(*
Nazwa:			GVL
Opis:			Zmienne wykorzystywane globalnie
Wersja:			v0.2
Data:			2021-10-05
Autor:			DP,DJ
Urzadzenia:		
Konfiguracja:	
Info:
*)

//{attribute 'qualified_only'}

VAR_GLOBAL
	(******MAIN**********)
	//Ogólne
	bFirstCycle										:BOOL;									// Zmienna pierwszego cyklu
	bManualMode										:BOOL; (**)								// Włączony tryb serwisowy
	tMachineCycleTime								:TIME;									// Czas cyklu maszyny
	bAddGlobalCounter								:BOOL;									// Pomocnicza do dodawania licznika przy odrzucie	
	bAddBadPackageReason							:BOOL;
	bAddBadPackageReason2							:BOOL;
	bChangeover										:BOOL;		
	bPhaseChanging									:BOOL;									// Zmiana trybu na dwufazowy
	bBottleSorterDisable							:BOOL:=FALSE;
	bCapSorterDisable								:BOOL:=FALSE;	
	bFastSpeed										:BOOL;
	
	//Resetowanie 
	bCycleReseting									:BOOL;									//Resetowanie cyklu, trwa 1 sek
	bAllStationDoneDelay							:BOOL;
	bHomingDialog									:BOOL;									//Wyświetl komunikat o bazowaniu
	bHomingCanceled									:BOOL;									// Anulowano bazowanie
	bHoming											:BOOL;									// Trwa bazowanie
	bFirstPositioningDone							:BOOL;
	bRecipeChangePositioning						:BOOL;
	sHomingText										:STRING;
	bResetAfterErrorOrEstop							:BOOL;
	bResetStates									:BOOL;									//Reset cyklu i formatek
	//CycleLogic
	bRobotStationDone								:BOOL;									// Skonczyło się dozowanie lub wyłaczone
	nCheckWeiginhForm								:BOOL;
	//nExitWheelFormsTime							:UINT;									// Czas na wypuszczenie formatki z karuzeli jak pracuje transporter
	
	//Rejestry przesuwne
	bRFIDChecker									:BOOL;									// Sprawdzanie RFID
	bRFIDClearAfterRobot							:BOOL;									// Usuwanie numeru RFID za robotem
	iRFIDClearNr1AfterRobot							:INT;									// Usuwanie numeru RFID za robotem, usuniety = 0
	iRFIDClearNr2AfterRobot							:INT;									// Usuwanie numeru RFID za robotem, usuniety = 0
		
	eClearPackageState								:S_PackageState;
	
	eBottleFeederPackageState						:ARRAY [1..17] OF S_PackageState;		// [1..2] Struktura pod podajnikiem butelek

	eBeforeGatePackageState							:ARRAY [1..17] OF S_PackageState;		// [1..2] Struktura przed szlabane
	eBeforeDispencersPackageState					:ARRAY [1..17] OF S_PackageState;		// [1..4] Struktura przed dozownikami
	eDispencersPackageState							:ARRAY [1..17] OF S_PackageState;		// [1..4] Struktura pod dozownikami
	eAfterDispencersPackageState					:ARRAY [1..17] OF S_PackageState;		// [1..4] Struktura za dozownikami 
	eWeightPackageState								:ARRAY [1..17] OF S_PackageState;		// [1..5] Struktura nad wagami

	eBeforeLidFeeder2PackageState					:ARRAY [1..17] OF S_PackageState;		// [] Struktura przed podawaniem platynek
	eBeforeLidFeederPackageState					:ARRAY [1..17] OF S_PackageState;		// [] Struktura przed podawaniem platynek
	eLidFeederPackageState							:ARRAY [1..17] OF S_PackageState;		// [] Struktura podawania platynek
	eAfterLidFeederPackageState						:ARRAY [1..17] OF S_PackageState;		// [] Struktura przed podawaniem platynek
	eBeforeLidSealerPackageState					:ARRAY [1..17] OF S_PackageState;		// [] Struktura przed zgrzewaniem platynek
	eLidSealerPackageState							:ARRAY [1..17] OF S_PackageState;		// [] Struktura zgrzewanie platynek
	
	eBeforeGateCapSorterPackageState				:ARRAY [1..17] OF S_PackageState;		// [1..4] Struktura przed RFID sortera nasadek
	eBeforeCapSorterPackageState					:ARRAY [1..17] OF S_PackageState;		// [1..4] Struktura przed sorterem
	eCapSorterPackageState							:ARRAY [1..17] OF S_PackageState;		// [1..4] Struktura pod sorterem
	eAfterCapSorterPackageState						:ARRAY [1..17] OF S_PackageState;		// [1..4] Struktura za sorterem
	eBeforeCapControlPackageState					:ARRAY [1..17] OF S_PackageState;		// [1..1] Struktura pod sprawdzaniem obecnosci nakretki
	eBeforeScrewersPackageState						:ARRAY [1..17] OF S_PackageState;		// [1..6] Struktura przed zakręcarkami 
	eBeforeScrewers2PackageState					:ARRAY [1..17] OF S_PackageState;		// [1..6] Struktura przed zakręcarkami przed czujnikiem
	eUnderScrewerPackageState 						:ARRAY [1..17] OF S_PackageState;		// [1..3] Struktura pod zakręcarkami 
	eAfterScrewerPackageState						:ARRAY [1..17] OF S_PackageState;		// [1..8] Struktura za zakręcarkami 
	eUnderCorrectCapPackageState					:ARRAY [1..17] OF S_PackageState;		// [1..7] Struktura pomiedzy robotem a sprawdzeniem poprawnego zakrecenia
	eUnderCorrectCapPackageStateTemp				:ARRAY [1..17] OF S_PackageState;		// [1..7] Struktura pomiedzy robotem a sprawdzeniem poprawnego zakrecenia	
	eRobotPackageState								:ARRAY [1..17] OF S_PackageState;		// [1..2] Struktura pod robotem
	eHistoryPackageState							:ARRAY [1..1000] OF S_PackageState;		// Struktura historyczna przetransferowanych butelek
	eTempState1										:ARRAY [1..17] OF S_PackageState;		// [1..12] Za waga
	eTempState2										:ARRAY [1..17] OF S_PackageState;		// [1..12] Za podajnikiem butelek
	eTempState3										:ARRAY [1..17] OF S_PackageState;		// [1..12] Za sorterem nakretek	
	eRobotTempState									:ARRAY [1..17] OF S_PackageState;    	//  Pod robotem

	// Dodatkowe rejestry przy dozowaniu dwufazowyn
	
	eWeightPackage2PhasePackageState				:ARRAY [1..17] OF S_PackageState;		// [1..5] Struktura nad wagami (** dodane 07.04.2022**)
	eBeforeDispencer34PackageState2Phase			:ARRAY [1..17] OF S_PackageState;		// [1..5] Struktura nad wagami (** dodane 07.04.2022**)
	eDispencer34PackageState2Phase					:ARRAY [1..17] OF S_PackageState;		// [1..5] Struktura nad wagami (** dodane 07.04.2022**)
	eAfterDispencer34PackageState2Phase				:ARRAY [1..17] OF S_PackageState;		// [1..5] Struktura nad wagami (** dodane 07.04.2022**)
	eBeforeDispencer12PackageState2Phase			:ARRAY [1..17] OF S_PackageState;		// [1..5] Struktura nad wagami (** dodane 07.04.2022**)
	eDispencer12PackageState2Phase					:ARRAY [1..17] OF S_PackageState;		// [1..5] Struktura nad wagami (** dodane 07.04.2022**)
	eAfterDispencer12PackageState2Phase				:ARRAY [1..17] OF S_PackageState;		// [1..5] Struktura nad wagami (** dodane 07.04.2022**)

	(******P00_Alarms*****)

	AbActiveWarningDescription								:ARRAY [0..63] OF BOOL;	//  Aktywne ostrzeżenia	
	
	//Sygnał dzwiekowy
	bSoftAlarm										:BOOL;
	
	bResetError										:BOOL:=FALSE;(**)						// Zmienna resetująca stację/błąd w PLC ,wystawia się po wciśnięciu ResetVisuCmd			
	//Reset Diagnostyki	
	
	//Alarmy inne*
	GeneralAlarms									:S_Error;								// 1 Ogólne
	//*Alarmy Stacji
	FormTransporterDispencerError					:S_Error;								// 2 Transporter wwjazdowy pod dozowniki
	FormTransporterScrewerError						:S_Error;								// 2 Transporter wyjściowy
	FormTransporterROPPError						:S_Error;
	FormTransporterAfterCapSorterError				:S_Error;
	FormTransporterBeforeScrewerError				:S_Error; 								// 3 Transporrter przed zakręcarkami
	FormTransporterSlowerError						:S_Error; 								// Spowalniacz
	FormTransporterAfterScrewerError				:S_Error; 								// 3 Transporrter przed zakręcarkami
	FormTransporterAfterBottleTransferError			:S_Error; 								
	BottleFeederError								:S_Error;								// Podajnik butelek
	BottleFeederTurnTableError						:S_Error;								// Stół obrotowy podajnika butleek
	BottleFeederFormGateError						:S_Error;								// Stoper formatek
	PucksInserterError								:S_Error;								// Podajnik butelek
	PucksInserterTurnTableError						:S_Error;								// Stół obrotowy podajnika opakowań
	PucksInserterFormGateError						:S_Error;								// Stoper formatek
	PucksInserterPushTableError_m1					:S_Error;								//71U3
	PucksInserterPushTableError_m2					:S_Error;								//71U4
	PucksInserterPushTableError_m3					:S_Error;								//
	GateBeforeDispencersError						:S_Error;		   						// 3A Szlaban przed dozownikami
		

	BarrierBetweenDispencers						:S_Error;								// Obsługa błędów szlaban dozowniki ( dozowanie dwufazowe, pod dozownikamia);
	BarrierBetweenWeights							:S_Error;								// Obsługa błędów stacji szlabanu pomiedzy wagamia ( dozowanie dwufazowe, wjazd na wagi);
	
	// Alarm wyciągu
	
	ExhaustFanError									:S_Error;
	SensorAcetoneError								:S_Error;								// Obśługa błedów czujnika acetonu
	SensorAirFlowError								:S_Error;								// Obsługa błędów czujnika przepływu 
	
	BottlePusherError								:S_Error;	
	//DispencerGatesError							:S_Error;								// 4 Szlabany pod dozownikami
	DispencersDragLeftError							:S_Error;								// Przeciąganie formatek
	DispencersDragRightError						:S_Error;								// Przeciąganie formatek (** 15.04.22 Damian**)
	

	DispencersCatch1Error							:S_Error;								// 4 Chwytak butelek dozownika 1
	DispencersCatch2Error							:S_Error;								// 4 Chwytak butelek dozownika 2
	DispencersCatch3Error							:S_Error;								// 4 Chwytak butelek dozownika 3
	DispencersCatch4Error							:S_Error;								// 4 Chwytak butelek dozownika 4
	Dispencer1Error									:S_Error;								// 5 Dozownik nr 1
	Dispencer2Error									:S_Error;								// 6 Dozownik nr 2
	Dispencer3Error									:S_Error;								// 6 Dozownik nr 3	
	Dispencer4Error									:S_Error;								// 6 Dozownik nr 4		
	TankHeatingError								:S_Error;								// Grzanie zbiornka

	WeightLiftError									:S_Error;
	
	Weight1Error									:S_Error;								// 8 Waga pierwsza jednofazowe
	Weight2Error									:S_Error;								// 8 Waga druga jednofazowe
	Weight3Error									:S_Error;								// 8 Waga trzecia jednofazowe
	Weight4Error									:S_Error;								// 8 Waga czwarta jednofazowe
	Weight5Error									:S_Error;								// 8 Waga piąta jednofazowe   	(** dodane 07.04.2022**)
	Weight6Error									:S_Error;								// 8 Waga szósta jednofazowe	(** dodane 07.04.2022**)
	
	
	GateAfterWeightError							:S_Error;								// 9 Szlaban za wagamia
		
	Dispencer1CorrectionError						:S_Error;	
	Dispencer2CorrectionError						:S_Error;
	Dispencer3CorrectionError						:S_Error;	
	Dispencer4CorrectionError						:S_Error;	
	WickFeederSorterError							:S_Error;
	
	
	CapFeederError									:S_Error;								// 14 
	CapSorterDragError								:S_Error;								// 15  Przeciąganie pod sorterem nasadek
			
	CapPuttedCheckError								:S_Error;								// 17 Wykrycie zakrętki
	
	GripperScrewerCatch1Error						:S_Error;								// 18 Chwytak zakręcarki szczękowej
	GripperScrewerCatch2Error						:S_Error;								// 18 Chwytak zakręcarki szczękowej
	GripperScrewer1Error							:S_Error;								// 19 Zakręcerka szczękowa 1
	GripperScrewer2Error							:S_Error;								// 19 Zakręcerka szczękowa 1

	BottleDragError									:S_Error;								//19.1 Przeciąganie butelek pod zakręcarkami
	CapCorrectCheckError							:S_Error;								// 21B Sprawdzanie zakręconej nakrętki
	CapCorrectCheckCameraError						:S_Error;
	BottleTransferError								:S_Error;								// 22 Robot
	GateRobotError									:S_Error;								// 22 Szlabany pod robotem
	BottleTransferAfterDragError					:S_Error;								// 14 

	BadBottleConveyorError							:S_Error;								// 23 Transporter odrzuconych butelek	
	LabelMachineError								:S_Error;								// 24 Etykieciarka
	TanksError										:S_Error;								// 24 Zbiorniki
	ExitTurnTableError								:S_Error;								// 25 Stół odbierający
	ExitConveyorError								:S_Error;								// 


	BarrierLidFeeder								: S_Error;								// Podajnik platynek 
	LidFeederError									: S_Error;								// Podajnik platynek 
	LidFeeder2Error									: S_Error;								// Podajnik platynek 2
	LidFeederFormPositioningError					: S_Error;	
						
	BarrierWickFeeder								: S_Error;
	WickFeederDragError								: S_Error;
	WickFeederError									: S_Error;
	WickFeeder2Error								: S_Error;
	WickFeederFormPositioningError					: S_Error;
	
	LidFeederDragError								: S_Error;								// Przeciąganie formatek                                                                                          
	LidPuttedCheckError								: S_Error;								// Wykrycie platynki                                                                                         
	LidSealerError									: S_Error;								// Zgrzewarka 1
	LidSealer2Error									: S_Error;								// Zgrzewarka 2
	LidSealerDragError								: S_Error;								// Przeciąganie formatek
	
	
	
	
	//Warningi
	TanksWarning									:ARRAY [0..7] OF S_Warning;							
	BottleTransferWarning							:ARRAY [0..7] OF S_Warning;	
	GeneralWarning1									:ARRAY [0..7] OF S_Warning;
	WeightWarning									:ARRAY [0..7] OF S_Warning;		
	DispencersWarning								:ARRAY [0..7] OF S_Warning;		
	ScrewersWarning									:ARRAY [0..7] OF S_Warning;		
	BottleFeederWarning								:ARRAY [0..7] OF S_Warning;
	ExSensorWarning									:ARRAY [0..7] OF S_Warning;
	CapFeederWarning								:ARRAY [0..7] OF S_Warning;	
	CapSorterWarning								:ARRAY [0..7] OF S_Warning;		
	BottleSorterWarning								:ARRAY [0..7] OF S_Warning;	
	LidFeederWarning								:ARRAY [0..7] OF S_Warning;		
	WickFeederWarning								:ARRAY [0..7] OF S_Warning;	
	WickFeederSorterWarning							:ARRAY [0..7] OF S_Warning;	
	(********P00_OEE********)		
	udiCounterExecuteTimeTemp						:UDINT;
	udiCounterErrorTimeTemp							:UDINT;
	udiCounterReadyTimeTemp							:UDINT;

	
	(******P00_Basic*******)
	//impulsy
	bImp1Sec										:BOOL;									// Impuls na zbocze generatora 1 sek
	b1Hz											:BOOL;									// Generator 1 sekundowy
	bV1Hz											:BOOL;									// bit o czest. 1Hz
	b2Hz											:BOOL;									// Generator 0,5 sekundowy
	//czas
	dtActTime										:DT;
	wYear 											:WORD;
	wMonth											:WORD;
	wDayOfWeek 										:WORD;
	wDay 											:WORD;
	wHour 											:WORD;
	wMinute 										:WORD;
	wSecond 										:WORD;
	wMilliseconds 									:WORD;

	//Zmienne podst.
	bAlwaysFalse									:BOOL:=FALSE;							//Zawsze zero
	
	(*****P00_PneumaticsValves***)
	(*****Receptury****)	
	bVTEMEnable										:BOOL;
	lrGripperScrewerPressure						:LREAL;									//Ciśnienie siłownika chwytaka nasadki zakręcarki szczękowej 1 (0.0 kg)
	lrGripperScrewerPressureExhaustLevel			:LREAL;									//Prędkość zamykania siłownika chwytaka nasadki zakręcarki szczękowej 1 (0.0-100.0 %)
	lrGripperScrewerCatchPressure					:LREAL;									//Ciśnienie siłownika chwytaka butelki zakręcarki szczękowej 1 (0.0 kg)
	lrGripperScrewerCatchPressureExhaustLevel		:LREAL;									//Prędkość zamykania siłownika chwytaka butelki zakręcarki szczękowej 1 (0.0-100.0 %)
	lrDispencerCatchPressure						:LREAL;

	(*****P0_Recipes***)
	(*****Receptury****)
	sRecipeName										:STRING;				
	sRecipeIndex									:STRING;				
	nRecipeIndex									:REAL;					
	bRecipeAfterPowerStateChosen					:BOOL;									//Receptura w stanie Power została wybrana (Pierwsza receptura po uruchomieniu)
	iPackageCapType									:INT; 									// Typ nasadki 
	iPackageCapDiameter								:INT;
	
	//[H] Praca w trybie wybuchowym
	bExEnable										:BOOL;						// [H] Tryb EX
	
	
	(****P01_BottleFeeder****)
	bBottleFeederEnable								:BOOL;									// Zezwolenie na pracę stacji podawania opakowań
	bBottleFeederDoHoming							:BOOL;									// Wykonanie bazowania stacji podawania butelek
	bBottleFeederTurnTableRun						:BOOL;									// Komenda startu stołu obrotwego
	iBottleFeederBottleSensorDelay					:INT;
	iBottleFeederFormGateDelay						:INT;
	iBottleFeederAllowFormDelay						:INT;
	bBottleFeederFormGateRun						:BOOL;									// Bit sterujacy działanie bramki 
	iBottleFeederTurntableVelocitySV				:UDINT;	

	(****P01_PucksInserter****)
	bPucksInserterEnable							:BOOL;									// Zezwolenie na pracę stacji 
	bPucksInserterDoHoming							:BOOL;									// Wykonanie bazowania stacji 
	bPucksInserterTurnTableRun						:BOOL;									// Komenda startu stołu obrotwego
	iPucksInserterBottleSensorDelay					:INT;
	iPucksInserterFormGateDelay						:INT;
	iPucksInserterFormGateDelayAdd					:INT;	
	iPucksInserterAllowFormDelay					:INT;
	bPucksInserterFormGateRun						:BOOL;									// Bit sterujacy działanie bramki 
	iPucksInserterTurntableVelocitySV				:UDINT;	
	iPucksInserterConveyorVelocitySV				:UDINT;	
	aPucksInserterWheelAxisRef						:AXIS_REF;								// Struktura osi 
	lrPucksInserterWheelOffset						:LREAL;									// Offset karuzeli +-10 st.
	lrPucksInserterWheelAcceleration				:LREAL;									// Przyspieszenie 
	lrPucksInserterWheelVelocity					:LREAL;									// Prędkość 
	lrPucksInserterHammerHeightSV					:LREAL;									// Pozycja
	
	//Push table 27.05 Vasyl	
	bPucksInserterPushTable_m1_Enable					:BOOL;
	bPucksInserterPushTable_m1_Run						:BOOL;
	udiPucksInserterPushTable_m1_VelocitySV				:UDINT;
	bPucksInserterPushTable_m2_Enable					:BOOL;
	bPucksInserterPushTable_m2_Run						:BOOL;
	udiPucksInserterPushTable_m2_VelocitySV				:UDINT;
	bPucksInserterPushTable_m3_Enable					:BOOL;
	bPucksInserterPushTable_m3_Run						:BOOL;
	udiPucksInserterPushTable_m3_VelocitySV				:UDINT;

	udiPucksInserterPushTableActuatorPUSHDelay			:UDINT;
	udiPucksInserterPushTableActuatorPULLDelay			:UDINT;
	udiPucksInserterPushTableOFFDelay					:UDINT;

	(****P01_BottleSorter****)
	//Po komunikacji
	
	(*****P01_Gates********)
	bGateBeforeDispencersEnable						:BOOL;									//Zezwolenie na pracę szlabanów pod robotem
	nGateBeforeDispencersTimeFormInserting			:UINT;									//Czas od momentu wjazdu formatek do zamkniecia 1 szlabanu pod robotem
	
	bGateAfterWeightEnable							:BOOL;									//Zezwolenie na pracę szlabanów pod robotem
	nGateAfterWeightTimeFormInserting				:UINT;									//Czas od momentu wjazdu formatek do zamkniecia 1 szlabanu pod robotem
		
	bBarrierLidFeederEnable							:BOOL;									//Zezwolenie na pracę szlabanów pod robotem
	nBarrierLidFeederTimeFormInserting				:UINT;									//Czas od momentu wjazdu formatek do zamkniecia 1 szlabanu pod robotem
	
	bGateRobotEnable								:BOOL;									//Zezwolenie na pracę szlabanów pod robotem
	nGateRobotTimeFormInserting						:UINT;									//Czas od momentu wjazdu formatek do zamkniecia 1 szlabanu pod robotem
	
	(*****P01_Barriers********)
	bBarrierWeightRun								:BOOL;									// Komenda otwarcia bariery przed wagami
	bBarrierDispencerRun							:BOOL;									// Komenda otwarcia bariery przed wagami
	
	(*****P02_Dispencers***)
	bCIP											: BOOL; // Włączone mycie CIP
	bDispencer1Cleaning								: BOOL;	// Mycie dozowników
	bDispencer2Cleaning								: BOOL;	// Mycie dozowników
	bDispencer3Cleaning								: BOOL;	// Mycie dozowników
	bDispencer4Cleaning								: BOOL;	// Mycie dozowników

	bDispencer1DoSync								: BOOL;	// Ustawienie tłoka/podnośnika 1 dozownika na konkretną pozycję (otwierają się zawory ssania) tylko w trybie serwisowym 
	bDispencer2DoSync								: BOOL;	// Ustawienie tłoka/podnośnika 2 dozownika na konkretną pozycję (otwierają się zawory ssania) tylko w trybie serwisowym 
	bDispencer3DoSync								: BOOL;	// Ustawienie tłoka/podnośnika 3 dozownika na konkretną pozycję (otwierają się zawory ssania) tylko w trybie serwisowym 
	bDispencer4DoSync								: BOOL;	// Ustawienie tłoka/podnośnika 4 dozownika na konkretną pozycję (otwierają się zawory ssania) tylko w trybie serwisowym 

	//Dozowniki 
	bDispencer12AllowDosingAfterDrag				:BOOL;
	bDispencer34AllowDosingAfterDrag				:BOOL;	
	bDoorDispencerOpen								:BOOL;
	bDosingTwoPhases								:BOOL;									//Dozowanie dwu fazowe
	bDispencersDoHoming								:BOOL;									//Wykonanie bazowania dozowniki
    lrDispencersLifterReadyPosition					:LREAL;									//Pozycja podnonika przy której dozowniki są w stanie gotowości
	uiDispencerStartDosingDelay						:UINT;(*0-3000*)				 		// Czas opóźnienia rozpoczęcia dozowania

//	Dozownik 1
	aDispencer1AxisRef								:AXIS_REF;//ActPos	(**)				// Struktura osi dozownika 1
	aDispencerLifter12AxisRef						:AXIS_REF;//ActPos	(**)				// Struktura osi dozownika 1
	bDispencer1Enable								:BOOL; 									// Zezwolenie na prace dozownika 1
	lrDispencer1DoseVolume							:LREAL:=195; 							// Objętoć do wydozowania przez dozownik 1
	bDispencer1LiftSynchroPh1						:BOOL;						 			// Polecenie synchronizacji dozownika z podnonikiem w fazie 1 Dozownika 1
	bDispencer1LiftSynchroPh2						:BOOL; 					 				// Polecenie synchronizacji dozownika z podnonikiem w fazie 2 Dozownika 1
	bDispencer1LiftSynchroPh3						:BOOL; 									// Polecenie synchronizacji dozownika z podnonikiem w fazie 3 Dozownika 1
	lrDispencer1Phase1Volume						:LREAL:=100;							// Objętoć do której ma trwać faza pierwsza dozowania dozownika 1
	lrDispencer1Phase2Volume						:LREAL:=100;							// Objętoć do której ma trwać faza druga dozowania dozownika 1
	lrDispencer1Phase1Velocity						:LREAL:=500;							// Prędkoć z jakš ma byc wykonywana faza pierwsza dozowania dozownika 1
	lrDispencer1Phase2Velocity						:LREAL:=500;							// Prędkoć z jakš ma byc wykonywana faza druga dozowania dozownika 1
	lrDispencer1Phase3Velocity						:LREAL:=500;							// Prędkoć z jakš ma byc wykonywana faza trzecia dozowania dozownika 1
	lrDispencer1SuckVelocity						:LREAL:=500;							// Prędkoć z jakš ma byc wykonywane zasysanie dozownika 1
	lrDispencer1Phase1Acceleration					:LREAL:=3000;							// Przyspieszenie z jakim ma byc wykonywana faza 1  dozownika 1
	lrDispencer1Phase2Acceleration					:LREAL:=3000;							// Przyspieszenie z jakim ma byc wykonywana faza 2  dozownika 1
	lrDispencer1Phase3Acceleration					:LREAL:=3000;							// Przyspieszenie z jakim ma byc wykonywana faza 3  dozownika 1
	lrDispencer1SuckAcceleration					:LREAL:=3000;							// Przyspieszenie z jakim ma byc wykonywane zasysanie dozownika 1
	lrDispencer1Phase1Deceleration					:LREAL:=3000;							// Zwalnianie z jakim ma byc wykonywana faza 1  dozownika 1
	lrDispencer1Phase2Deceleration					:LREAL:=3000;							// Zwalnianie z jakim ma byc wykonywana faza 2  dozownika 1
	lrDispencer1Phase3Deceleration					:LREAL:=3000;							// Zwalnianie z jakim ma byc wykonywana faza 3  dozownika 1
	udiDispencer1DosingDoneDelayTime				:UDINT:=20; 							// Opóźnienie wykonania cyklu dozy przez dozownik 1 [ms]
	lrDispencer1SuckValveOpenVolume					:LREAL:=0;(*Z 0-15*)					//[3] Objętość przy której ma byc otwierany zawór ssania dozownika 1
	lrDispencer1SuckValveOpenTimeDelay				:LREAL:=0;(*NOWA 0-1000*)				// [3] Opóżnienie rozpoczęcia ssania po tłoczeniu [ms]
	lrDispencer1SuckValveCloseVolume				:LREAL:=0;(*Z 0-15*)					// [4] Objętość przy której ma byc zamykany zawór ssania dozownika 1
	lrDispencer1SuckValveCloseTimeDelay				:LREAL:=0;(*NOWA 0-2000*)				// [4] Opóżnienie zamknięcia zaworu ssącego [ms]
	lrDispencer1DoseValveOpenVolume					:LREAL:=0;(*Z 0-15*)					//[1] Objętość przy której ma byc otwierany zawór tłoczenia (iglica) dozownika 1 
	lrDispencer1DoseValveOpenTimeAcc				:LREAL:=0;(*NOWA 0-500*)				// [1] Przyśpieszenie otwarcia zaworu tłoczenia [ms]
	lrDispencer1DoseValveCloseVolume				:LREAL:=0;(*0-15*)						// [2] Objętość przy której ma byc zamykany zawór tłoczenia (iglica) dozownika 1 
	lrDispencer1DoseValveCloseTimeDec				:LREAL:=0;(*NOWA 0-1000*)				// [2] Opóźnienie zamknięcia zaworu tłoczenia [ms]
	lrDispencer1DoseSuckingVolume					:LREAL:=0;(*NOWA 0-100*)			  	//[5] [Podsysanie] Wartość dozy do posysenia [ml]	
	lrDispencer1DoseSuckingTimeDelay				:LREAL:=0;(*NOWA 0-500*)  				//[6] [Podsysanie] Opóźnienie podsysania [ms]
	bDispencer1DoseSucking							:BOOL;(*NOWA*) 					 		// [Podsysanie] Opcja podsysania przy dozowaniu
	lrDispencer1LifterStartDosePosition				:LREAL:=20;								// Pozycja podnonika przy której rozpoczyna sie dozowanie dozownika 1
	lrDispencer1LifterStopDosePosition				:LREAL:=60;								// Pozycja podnonika przy której kończy sie dozowanie dozownika 1
	lrDispencer1LifterVelocity						:LREAL:=20;								// Prędkoć podnonika dozownika 1	
	lrDispencer1LifterAcceleration					:LREAL:=2;								// Przyspieszenie podnonika dozownika 1
	lrDispencer1LifterDeceleration					:LREAL:=2;								// Przyspieszenie podnonika dozownika 1

//	Dozownik 2
	aDispencer2AxisRef								:AXIS_REF;//ActPos(**)					// Struktura osi dozownika 2
	bDispencer2Enable								:BOOL; 									// Zezwolenie na prace dozownika 2
	lrDispencer2DoseVolume							:LREAL:=195; 							// Objętoć do wydozowania przez dozownik 2
	bDispencer2LiftSynchroPh1						:BOOL;						 			// Polecenie synchronizacji dozownika z podnonikiem w fazie 1 Dozownika 2
	bDispencer2LiftSynchroPh2						:BOOL; 					 				// Polecenie synchronizacji dozownika z podnonikiem w fazie 2 Dozownika 2
	bDispencer2LiftSynchroPh3						:BOOL; 									// Polecenie synchronizacji dozownika z podnonikiem w fazie 3 Dozownika 2
	lrDispencer2Phase1Volume						:LREAL:=100;							// Objętoć do której ma trwać faza pierwsza dozowania dozownika 2
	lrDispencer2Phase2Volume						:LREAL:=100;							// Objętoć do której ma trwać faza druga dozowania dozownika 2
	lrDispencer2Phase1Velocity						:LREAL:=500;							// Prędkoć z jakš ma byc wykonywana faza pierwsza dozowania dozownika 2
	lrDispencer2Phase2Velocity						:LREAL:=500;							// Prędkoć z jakš ma byc wykonywana faza druga dozowania dozownika 2
	lrDispencer2Phase3Velocity						:LREAL:=500;							// Prędkoć z jakš ma byc wykonywana faza trzecia dozowania dozownika 2
	lrDispencer2SuckVelocity						:LREAL:=500;							// Prędkoć z jakš ma byc wykonywane zasysanie dozownika 2
	lrDispencer2Phase1Acceleration					:LREAL:=3000;							// Przyspieszenie z jakim ma byc wykonywana faza 1  dozownika 2
	lrDispencer2Phase2Acceleration					:LREAL:=3000;							// Przyspieszenie z jakim ma byc wykonywana faza 2  dozownika 2
	lrDispencer2Phase3Acceleration					:LREAL:=3000;							// Przyspieszenie z jakim ma byc wykonywana faza 3  dozownika 2
	lrDispencer2SuckAcceleration					:LREAL:=3000;							// Przyspieszenie z jakim ma byc wykonywane zasysanie dozownika 2
	lrDispencer2Phase1Deceleration					:LREAL:=3000;							// Zwalnianie z jakim ma byc wykonywana faza 1  dozownika 2
	lrDispencer2Phase2Deceleration					:LREAL:=3000;							// Zwalnianie z jakim ma byc wykonywana faza 2  dozownika 2
	lrDispencer2Phase3Deceleration					:LREAL:=3000;							// Zwalnianie z jakim ma byc wykonywana faza 3  dozownika 2
	udiDispencer2DosingDoneDelayTime				:UDINT:=20; 							// Opóźnienie wykonania cyklu dozy przez dozownik 2 [ms]
	lrDispencer2SuckValveOpenVolume					:LREAL:=0;(*Z 0-15*)					// [3] Objętość przy której ma byc otwierany zawór ssania dozownika 2
	lrDispencer2SuckValveOpenTimeDelay				:LREAL:=0;(*NOWA 0-1000*)				// [3] Opóżnienie rozpoczęcia ssania po tłoczeniu [ms]
	lrDispencer2SuckValveCloseVolume				:LREAL:=0;(*Z 0-15*)					// [4] Objętość przy której ma byc zamykany zawór ssania dozownika 2
	lrDispencer2SuckValveCloseTimeDelay				:LREAL:=0;(*NOWA 0-2000*)				// [4] Opóżnienie zamknięcia zaworu ssącego [ms]
	lrDispencer2DoseValveOpenVolume					:LREAL:=0;(*Z 0-15*)					// [1] Objętość przy której ma byc otwierany zawór tłoczenia (iglica) dozownika 2 
	lrDispencer2DoseValveOpenTimeAcc				:LREAL:=0;(*NOWA 0-500*)				// [1] Przyśpieszenie otwarcia zaworu tłoczenia [ms]
	lrDispencer2DoseValveCloseVolume				:LREAL:=0;(*0-15*)						// [2] Objętość przy której ma byc zamykany zawór tłoczenia (iglica) dozownika 2 
	lrDispencer2DoseValveCloseTimeDec				:LREAL:=0;(*NOWA 0-1000*)				// [2] Opóźnienie zamknięcia zaworu tłoczenia [ms]
	lrDispencer2DoseSuckingVolume					:LREAL:=0;(*NOWA 0-100*)  				// [5] [Podsysanie] Wartość dozy do posysenia [ml]	
	lrDispencer2DoseSuckingTimeDelay				:LREAL:=0;(*NOWA 0-500*)  				// [6] [Podsysanie] Opóźnienie podsysania [ms]
	bDispencer2DoseSucking							:BOOL;(*NOWA*)  						// [Podsysanie] Opcja podsysania przy dozowaniu
	lrDispencer2LifterStartDosePosition				:LREAL:=20;								// Pozycja podnonika przy której rozpoczyna sie dozowanie dozownika 2
	lrDispencer2LifterStopDosePosition				:LREAL:=60;								// Pozycja podnonika przy której kończy sie dozowanie dozownika 2
	lrDispencer2LifterVelocity						:LREAL:=20;								// Prędkoć podnonika dozownika 2	
	lrDispencer2LifterAcceleration					:LREAL:=2;								// Przyspieszenie podnonika dozownika 2
	lrDispencer2LifterDeceleration					:LREAL:=2;								// Przyspieszenie podnonika dozownika 2

	//	Dozownik 3
	aDispencer3AxisRef								:AXIS_REF;//ActPos	(**)				// Struktura osi dozownika 3
	aDispencerLifter34AxisRef						:AXIS_REF;//ActPos	(**)				// Struktura osi dozownika 3
	bDispencer3Enable								:BOOL; 									// Zezwolenie na prace dozownika 3								

	//	Dozownik 4
	aDispencer4AxisRef								:AXIS_REF;//ActPos				(**)	// Struktura osi dozownika 4
	bDispencer4Enable								:BOOL; 									// Zezwolenie na prace dozownika 4
		
	//Podonosnik chwytaka i tacki 1,2,3,4
	bDispencersCatchEnable								:BOOL; 									// Zezwolenie na pracę chwytaka butelek pod dozownikami 1
	bDispencersCatchMaxPressure							:BOOL;									// Zwiekszona siła chwytania
	bDispencersCatch1DoHoming							:BOOL;									// Wykonanie bazowania przez chwytak i tacke pod dozownikiem 1
	lrDispencersCatchHeightSV							:LREAL:=36;  					       	// Zadana wartoć pozycji bazowania stacji chwytania opakowania pod dozownikami
	bDispencersCatch2DoHoming							:BOOL;									// Wykonanie bazowania przez chwytak i tacke pod dozownikiem 2
	bDispencersCatch3DoHoming							:BOOL;									// Wykonanie bazowania przez chwytak i tacke pod dozownikiem 3
	bDispencersCatch4DoHoming							:BOOL;									// Wykonanie bazowania przez chwytak i tacke pod dozownikiem 4

    (*Wartości dla nowych czujników wykrywania butelki pod dozownikami*)
    (*Są zależne od szerokości szyjki i dlatego trzeba je zapamiętywać*)
    (*Kalibracja chwytaków w serwisie będzie nadpisywała te wartości*)
    (*Będzie się je zmieniało przez kalibracje więc widocznośc tylko ustawić dla serwisu*)
    lrDispencersCatch1ClosedValue                    	:LREAL;                        // Chwytak 1 | wartość kalibracji zamkniętego chwytaka
    lrDispencersCatch1OpenValue                      	:LREAL;                        // Chwytak 1 | wartość kalibracji otwartego chwytaka
    lrDispencersCatch2ClosedValue                    	:LREAL;                        // Chwytak 2 | wartość kalibracji zamkniętego chwytaka
    lrDispencersCatch2OpenValue                      	:LREAL;                        // Chwytak 2 | wartość kalibracji otwartego chwytaka
    lrDispencersCatch3ClosedValue                   	:LREAL;                        // Chwytak 3 | wartość kalibracji zamkniętego chwytaka
    lrDispencersCatch3OpenValue                     	:LREAL;                        // Chwytak 3 | wartość kalibracji otwartego chwytaka
    lrDispencersCatch4ClosedValue                   	:LREAL;                        // Chwytak 4 | wartość kalibracji zamkniętego chwytaka
    lrDispencersCatch4OpenValue                      	:LREAL;                        // Chwytak 4 | wartość kalibracji otwartego chwytaka
    (*Tolerancja dla chwytaków - dla operatora*)
    lrDispencersCatchTolerance                       	:LREAL;                        // Tolerancja szyjki butelki pod dozownikami [0-100%]      
	
	//Przeciąganie formatek
	aFormsDragingRightAxisRef							:AXIS_REF;								// Struktura osi napędu krokowego przeciągania	
	bFormsDragingRightEnable							:BOOL;									// Zezwolenie na pracę przeciągania 
	bFormsDragingRightDoHoming							:BOOL;									// Wykonanie bazowania przeciągania
	bFormsDragingRightHeightSet							:BOOL;									// Wykonanie bazowania przeciągania
	lrFormsDragingRightVelocity							:LREAL:=100;							// Prędkośc przeciągania
	lrFormsDragingRightAcceleration						:LREAL:=12;								// Przyspieszenie przeciągania
	lrFormsDragingRightDeceleration						:LREAL:=15;								// Hamowanie przeciągania
	bFormsDragingRightPrepareRun						:BOOL;
	bFormsDragingRightRunCheck							:BOOL;		
	//Przeciąganie formatek
	aFormsDragingLeftAxisRef							:AXIS_REF;								// Struktura osi napędu krokowego przeciągania
	bFormsDragingLeftEnable								:BOOL;									// Zezwolenie na pracę przeciągania 
	bFormsDragingLeftDoHoming							:BOOL;									// Wykonanie bazowania przeciągania
	bFormsDragingLeftHeightSet							:BOOL;									// Wykonanie bazowania przeciągania
	lrFormsDragingLeftVelocity							:LREAL:=100;							// Prędkośc przeciągania
	lrFormsDragingLeftAcceleration						:LREAL:=12;								// Przyspieszenie przeciągania
	lrFormsDragingLeftDeceleration						:LREAL:=15;								// Hamowanie przeciągania
	bFormsDragingLeftPrepareRun							:BOOL;
	iFormsDragingFormCounter							:INT;
	bFormsDragingLeftRunCheck							:BOOL;	
	
	//Zbiorniki
	bTank1MixerEnable								:BOOL;(**)   					  		// Załaczanie mieszadła zbiornikowego 1
	bTankHeatingEnable								:BOOL;								    // Zezwolenie na pracę
	iTankHeatingTempSV								:INT;	
	bTank1SupplyPumpEnable							:BOOL;(**) 								// Załaczanie pompy zasilajacej zbiornik 1
	bTank1PressureEnable							:BOOL;									// Włączanie Ciśnienia w zbiorniku 1
	bTank2SupplyPumpEnable							:BOOL;(**) 								// Załaczanie pompy zasilajacej zbiornik 2
	uTank1LevelSetpoint								:UINT;(*o*)								// Wartość zadana masy do czujnika poziomu w zbiorniku nr 1
	bTank1LevelSignalInvert							:BOOL;									// Odwróć sygnał z czujnika zbiornika pierwszego
	bTank2LevelSignalInvert							:BOOL;									// Odwróć sygnał z czujnika zbionirka drugiego
	uTank2LevelSetpoint								:UINT;(*o*)								// Wartość zadana masy do czujnika poziomu w zbiorniku nr 1
	//Zbiorniki-dodatkowe
	bTankRainbowMode								:BOOL;
	(*****P05_Weight*****)
	bWeightLiftEnable								:BOOL;	
	bWeightLiftDoHoming								:BOOL;
	bWeightLiftDeparture							:BOOL;
	bWeight1234ReleaseBlock							:BOOL;	
	bWeightLift2PhaseRun							:BOOL;
	bWeight56ReleaseBlock							:BOOL;	
	bWeighingAutoTarePreset							:BOOL;	
	bWeighingAutoTare								:BOOL;	
	
	bWeight1Enable									:BOOL;									// Zezwolenie na pracę wagi 1
	lrWeightMassSV									:LREAL;									// Waga zadana masy 
	lrWeight1Chart									:LREAL;									// Tylko do wykresów
	lrWeight2Chart									:LREAL;									// Tylko do wykresów
	lrWeight3Chart									:LREAL;									// Tylko do wykresów
	lrWeight4Chart									:LREAL;									// Tylko do wykresów
	lrWeight5Chart									:LREAL;									// Tylko do wykresów
	lrWeight6Chart									:LREAL;									// Tylko do wykresów
	
	iWeight1ActuatorUpDelay							:INT;									// Opóźnienie podnoszenia Waga 1	
	iWeight2ActuatorUpDelay							:INT;									// Opóźnienie podnoszenia Waga 2	
	iWeight3ActuatorUpDelay							:INT;									// Opóźnienie podnoszenia Waga 3	
	iWeight4ActuatorUpDelay							:INT;									// Opóźnienie podnoszenia Waga 4	
	iWeight5ActuatorUpDelay							:INT;									// Opóźnienie podnoszenia Waga 5	
	iWeight6ActuatorUpDelay							:INT;									// Opóźnienie podnoszenia Waga 6	
	iWeight56ActuatorUpAddDelay						:INT;									// Opóźnienie podnoszenia Waga 5	
	iWeight14ActuatorUpAddDelay						:INT;									// Opóźnienie podnoszenia Waga 5	

	//Podajnik knotów
	bWickFeederEnable								: BOOL;									// Zezwolenie na pracę podajnika platynek
	bWickFeederDoHoming								: BOOL;									// Bazowanie podajnika platynek
   lrWickFeederHeightPosSV							: LREAL := 72;							// Wysokoć na której ma znajdować się podajnik platynek

	//Przeciąganie podajnik knotów
	bWickFeederDragingStationEnable					: BOOL;
	bWickFeederDragingStationDoHoming				: BOOL;
	bWickFeederDragingStationPrepareRun				: BOOL;
	lrWickFeederDragingStationVelocity				: LREAL; 							// Zadana prędkosć ruchu przeciągania formatek pod zakręcarkam
	lrWickFeederDragingStationAcceleration			: LREAL;							// Przyspieszenie przeciągania
	lrWickFeederDragingStationDeceleration			: LREAL;							// Hamowanie przeciągania
	aWickFeederDragingAxisRef						: AXIS_REF;
	bWickFeederDragingHeightSet						: BOOL;	
	iWickFeederSorterTimeDelayOn					: INT;
	iWickFeederSorterTimeDelayOff					: INT;
	iWickFeederSorterTimeToEmptySleeveError			: INT;

	//Podajnik platynek
	bLidFeederEnable								: BOOL;									// Zezwolenie na pracę podajnika platynek
	bLidFeederDoHoming								: BOOL;									// Bazowanie podajnika platynek
    bLidFeederHeaterEnable							: BOOL;									// Zezwolenie na prace grzałki podajnika platynek
	iLidFeederHeatingTime							: INT 	:= 1000;						// Czas zgrzewania wstępnego podajnika platynek [ms]
    lrLidFeederHeightPosSV							: LREAL := 72;							// Wysokoć na której ma znajdować się podajnik platynek
    iLidFeeder1TempSV								: INT	:= 150;							// Temperatura zadana grzałki podajnika platynek
    iLidFeeder2TempSV								: INT	:= 150;							// Temperatura zadana grzałki podajnika platynek
	iLidFeederTempHisteresis						: INT;							 	  	// Histereza poprawnej temperatury grzałki (+/- *C), po jej przekroczeniu grzałka wpada w błšd
	bLidFeeder2Enable								: BOOL;									// Zezwolenie na pracę podajnika platynek	
	bLidFeederFormPositioningRun					: BOOL;	
	
	//Przeciąganie podajnik platynek
	bLidFeederDragingStationEnable					: BOOL;
	bLidFeederDragingStationDoHoming				: BOOL;
	bLidFeederDragingStationPrepareRun				: BOOL;
	lrLidFeederDragingStationVelocity				: LREAL; 							// Zadana prędkosć ruchu przeciągania formatek pod zakręcarkam
	lrLidFeederDragingStationAcceleration			: LREAL;							// Przyspieszenie przeciągania
	lrLidFeederDragingStationDeceleration			: LREAL;							// Hamowanie przeciągania
	aLidFeederDragingAxisRef						: AXIS_REF;
	bLidFeederDragingHeightSet						: BOOL;		                                                											
 													
	//Sprawdzanie platynek                          
   	bLidPuttedCheckDoHoming     					: BOOL;  								// Wykonanie bazowania stacji sprawdzania nakrętek
    bLidPuttedCheckEnable       					: BOOL;  								// Zezwolenie na prace stacji sprawdzania nakrętek
    lrLidPuttedCheckHeightSV 	 					: LREAL; 								// Wysokość na której ma znajdować się stacja sprawdzania nakrętek
	lrLidPuttedCheckPosition						: LREAL;								// Pozycja sprawdzania platynki
	lrLidPuttedCheckArea							: LREAL;								// Granicy sprawdzania platynki
	bLidPuttedCheckInCameraArea1					: BOOL;									// Wózek 1 sprawdzany
	bLidPuttedCheckInCameraArea2					: BOOL;									// Wózek 2 sprawdzany
	iLidPuttedCheckProgram							: INT;	
	
	//Przygrzewaczki
	lrLidSealerPressure								: LREAL;									//	Siła zgrzewania [kg]                                              
	//Przygrzewaczka 1                              
	bLidSealerEnable								: BOOL;									// Zezwolenie na pracę podajnika 
	bLidSealerDoHoming								: BOOL; 								// Wykonanie bazowania przez przygrzewacz platynek
    bLidSealerHeaterEnable							: BOOL;								    // Zezwolenie na prace grzałki 
    iLidSealerHeatingTime							: INT	:=700;						    // Czas zgrzewania  [ms]
    iLidSealer1TempSV								: INT	:=150;							// Temperatura zadana grzałki 
	nLidSealerTempHisteresis						: INT;							    	// Histereza poprawnej temperatury grzałki (+/- *C), po jej przekroczeniu grzałka wpada w błšd
    lrLidSealerHeightPosSV							: LREAL	:=55;						    // Wysokoć na której ma znajdować się grzałka
	                                                
	//Przygrzewaczka 2                              
    bLidSealer2Enable								: BOOL;									// Zezwolenie na pracę podajnika 								// Wykonanie bazowania przez przygrzewacz platynek 
	bLidSealer2HeaterEnable							: BOOL;								    // Zezwolenie na prace grzałki 
    iLidSealer2TempSV								: INT	:=150;							// Temperatura zadana grzałki 
	
	//Przeciąganie przygrzewaczka
	bLidSealerDragingStationEnable							: BOOL;
	bLidSealerDragingStationDoHoming				: BOOL;
	bLidSealerDragingStationPrepareRun				: BOOL;
	lrLidSealerDragingStationVelocity				: LREAL	:= 100; 						// Zadana prędkosć ruchu przeciągania formatek pod zakręcarkam
	lrLidSealerDragingStationAcceleration			: LREAL	:=12;							// Przyspieszenie przeciągania
	lrLidSealerDragingStationDeceleration			: LREAL	:=15;							// Hamowanie przeciągania
	aLidSealerDragingAxisRef						: AXIS_REF;
	bLidSealerDragingHeightSet						: BOOL;	
	iLidSealerDragFormCounter						: INT;
	
	//Przeciąganie za robotem (rotacja formatek)
	bAfterRobotDragingStationEnable							: BOOL;
	bAfterRobotDragingStationDoHoming				: BOOL;
	bAfterRobotDragingStationPrepareRun				: BOOL;
	lrAfterRobotDragingStationVelocity				: LREAL	:= 100; 						// Zadana prędkosć ruchu przeciągania formatek pod zakręcarkam
	lrAfterRobotDragingStationAcceleration			: LREAL	:=12;							// Przyspieszenie przeciągania
	lrAfterRobotDragingStationDeceleration			: LREAL	:=15;							// Hamowanie przeciągania
	aAfterRobotDragingAxisRef						: AXIS_REF;
	bAfterRobotDragingHeightSet						: BOOL;	
	iAfterRobotDragFormCounter						: INT;	
	
	(*****P05_WeightCorrection******)
	lrFormWeight 									:LREAL;									// Waga formatki
	
	lrFormWeight1RFID								:LREAL;									// Waga formatki z RFID
	lrFormWeight2RFID								:LREAL;									// Waga formatki z RFID
	lrFormWeight3RFID								:LREAL;									// Waga formatki z RFID
	lrFormWeight4RFID								:LREAL;									// Waga formatki z RFID
	
	lrFormWeight5RFID								:LREAL;									// Waga formatki z RFID
	lrFormWeight6RFID								:LREAL;									// Waga formatki z RFID

	lrMass1Density									:LREAL;(*#p*)							//Gęstoć masy [g/ml]
	lrMass2Density									:LREAL;(*#p*)							//Gęstoć masy [g/ml]
	lrCupWeight										:LREAL;(*#p*)							//Waga samego kubeczka [g]
	lrWholePackageWeight							:LREAL;(*#p*)							//Waga całego opakowania bez masy (kubeczek,platynka,nakrętka) [g]
	lrWeight1MeasurmentCorrection					:LREAL;(*#p*)							//Korekta wagi zmierzonej [g]//Korekta wagi zmierzonej [g]

	iWeightCorrectionNumberOfSamples				:UINT;									// Ilość próbek dla korekty dozy

	bDispencer1WeightCorrectionEnable				:BOOL;(*#p*)							//Zezwolenie na pracę bloku korekcji, jeli przełšczy sie w tryb 
	bDispencer2WeightCorrectionEnable				:BOOL;(*#p*)							//Zezwolenie na pracę bloku korekcji, jeli przełšczy sie w tryb 
	bDispencer3WeightCorrectionEnable				:BOOL;(*#p*)							//Zezwolenie na pracę bloku korekcji, jeli przełšczy sie w tryb 
	bDispencer4WeightCorrectionEnable				:BOOL;(*#p*)							//Zezwolenie na pracę bloku korekcji, jeli przełšczy sie w tryb 
	lrWeightUpperTolerance							:LREAL;(*#p*)							//Górny zakres tolerancji wagi [g]
	lrWeightLowerTolerance							:LREAL;(*#p*)							//Zakres tolerancji wagi poniżej zadanej [g]	

	(*****P08_CapFeeder*****)
	bCapFeederDoHoming: BOOL;										// Wykonanie bazowania stacji podajnika nakrętek
	bCapFeederEnable: BOOL; 	
    lrCapFeederHeightPosSV: LREAL;									 	
	iCapFeederTimeDelayOn: INT; 										
	iCapFeederTimeDelayOff: INT; 
	iCapFeederTimeToEmptySleeveError: INT;							// Czas do alarmu pustego rękawa 

	(*****P08_CapSorter*****)
	bCapFeederGateEnable	:BOOL;									// Załączenie szlabanu podawania zamknięć 
	iCapFeederGateBlockingTime	:INT;								// Czas blokowania szlabnu podawania zamknięć
	iCapFeederCheckCountNOK	:INT;									// Zliczanie butelek bez nasadek

	//Sorter nasadek
	bCapSorterOnlyWeightOKEnable				:BOOL;
	
	//Przeciąganie formatek
	aCapSorterDragAxisRef							:AXIS_REF;								// Struktura osi napędu krokowego przeciągania	
	bCapSorterDragEnable							:BOOL;									// Zezwolenie na pracę przeciągania 
	bCapSorterDragDoHoming							:BOOL;									// Wykonanie bazowania przeciągania
	bCapSorterDragHeightSet							:BOOL;									// Wykonanie bazowania przeciągania
	lrCapSorterDragVelocity							:LREAL:=100;							// Prędkośc przeciągania
	lrCapSorterDragAcceleration						:LREAL:=12;								// Przyspieszenie przeciągania
	lrCapSorterDragDeceleration						:LREAL:=15;								// Hamowanie przeciągania
	bCapSorterDragPrepareRun						:BOOL;
	iCapSorterDragFormCounter						:INT;
	
	(*****P09_CapPuttedCheck*****)
	bCapPuttedCheckDoHoming							:BOOL;									// Wykonanie bazowania stacji sprawdzania nakrętek
	bCapPuttedCheckEnable							:BOOL; 									// Zezwolenie na prace stacji sprawdzania nakrętek
	lrCapPuttedCheckHeightPosSV						:LREAL:=69;(**) 					   	// Wysokość na której ma znajdować się stacja sprawdzania nakrętek
	bCapPuttedCheckRun								:BOOL;
	
	(****P10A_BottleDrag****) 
	bBottleDragingStationEnable						:BOOL;
	lrBottleDragingStationVelocity					:LREAL; 				
	bBottleDragingStationDoHoming					:BOOL;
	bBottleDragingStationPrepareRun					:BOOL;
	aBottleDragingAxisRef							:AXIS_REF;				
	bBottleDragingHeightSet							:BOOL;						
	
	bDelay40sAfterReset								:BOOL;
	
	(*****P10_GripperScrewer********)
	aGripperScrewer1LiftAxisRef						:AXIS_REF;//ActPos						// Struktura NC napędu podnosnika zakręcarki szczękowej
	aGripperScrewer2LiftAxisRef						:AXIS_REF;//ActPos						// Struktura NC napędu podnosnika zakręcarki szczękowej
	aGripperScrewer1AxisRef							:AXIS_REF; 								// Struktura NC napędu zakręcarki szczękowej 1
	aGripperScrewer2AxisRef							:AXIS_REF; 								// Struktura NC napędu zakręcarki szczękowej 2
	aGripperScrewer1EncoderAxisRef					:AXIS_REF; 								// Struktura NC enkodera zakręcarki szczękowej 1
	aGripperScrewer2EncoderAxisRef					:AXIS_REF; 								// Struktura NC enkodera zakręcarki szczękowej 2
	bGripperScrewerDoHoming							:BOOL;(**)								// Bazowanie stacji zakręcarki szczękowej
	bGripperScrewer1Enable							:BOOL;						// Aktywacja pierwszeh zakrecarki
	bGripperScrewer2Enable							:BOOL;						// Aktywacja drugiej zakrecarki
	bGripperScrewerFindScrew						:BOOL; 						// Aktywacja szukania gwintu	
	lrGripperScrewerFindingScrewDegree				:LREAL; 					// Kąt szukania gwintu
	iGripperScrewer1Tool							:INT;						// Wybór narzędzia (1-5), opisy w tablicy AsGripperScrewerTool	
	bGripperScrewerOption1							:BOOL;						// Otwarty chwytak przy szukaniu gwintu
	bGripperScrewerOption2							:BOOL;						// Obrót do tyłu w pozycji dociskania
	bGripperScrewerOption3							:BOOL;						// Dodatkowe zamknięcie chwytakiem przed zakręceniem 
	bGripperScrewerOption4							:BOOL;						// Szukanie gwintu w pozycji dociskania
	bGripperScrewerOption5							:BOOL;						// Szukanie gwintu z czujnikiem wysokości
	bGripperScrewerOption6							:BOOL;						// Szukanie gwintu z czujnikiem wysokości
 	bGripperScrewerOption7							:BOOL;						// Szukanie gwintu z czujnikiem wysokości
 	lrGripperScrewerVelocity						:LREAL:=6000; 				// Prędkość zakręcania
	nGripperScrewerTightTime						:INT:=100;  				// Czas przytrzymania nakrętki z zadanym momentem [ms] 
	iGripperScrewerStartDelay						:INT;						// Zwoka przed zakręcaniem			
	lrGripperScrewingTightTorque					:LREAL;  					// Nastawa momentu zakręcania [Nm]
	lrGripperScrewing2TightTorque					:LREAL;  					// Nastawa momentu zakręcania 2[Nm]
	lrGripperScrewerReadyPosition					:LREAL := 250;  			// Pozycja gotowości
	lrGripperScrewerPushingCapPosition				:LREAL := 250;  			// Pozycja docisku nakrętki 
    lrGripperScrewerScrewingCapPosition				:LREAL := 250;  			// Pozycja zakręcania nakrętki
	lrGripperScrewerFindScrewPosition				:LREAL := 250;  			// Pozycja zakręcania nakrętki
	bGripperScrewerFindScrewAdjust					: BOOL; 								// Wlaczanie dłuższego szukania  z szukaniem MIN i MAX wysokości z czujnikiem wysokości 
	lrGripperScrewerTurnoversToFullScrewed 			:LREAL;
   	lrGripperScrewerThreadPitch						:LREAL;
	lrGripperScrewerThreadTimes						:LREAL;
	
	//Chytak zakrecarki
	bGripperScrewerCatch1Homing						:BOOL;
	bGripperScrewerCatch2Homing						:BOOL;
	
	bGripperScrewerCatch1DoHoming					:BOOL;(**)								// Bazowanie stacji łapania pod zakręcarki szczękowej
	bGripperScrewer1Catch							:BOOL;  						        // Rozkaz chwytania opakowania pod zakręcarkš
	nGripperScrewerCatchHeightSV					:LREAL:=36;(*#pp*)						// Zadana wartoć pozycji bazowania stacji chwytania opakowania pod zakręcarkš

	bGripperScrewerCatch2DoHoming					:BOOL;(**)								// Bazowanie stacji łapania pod zakręcarki szczękowej
	bGripperScrewer2Catch							:BOOL;  						        // Rozkaz chwytania opakowania pod zakręcarkš	
	
	(*****P11B_CapPuttedCheck*****)
	bCapCorrectCheckDoHoming						:BOOL;									// Wykonanie bazowania stacji sprawdzania nakrętek
	bCapCorrectCheckEnable							:BOOL; 									// Zezwolenie na prace stacji sprawdzania nakrętek
	lrCapCorrectCheckHeightPosSV					:LREAL:=69;(**) 				   		// Wysokość na której ma znajdować się stacja sprawdzania nakrętek
	bCapCorrectCheckCameraEnable					:BOOL;  
	iCapCorrectCheckCameraProgram                   :INT;	
	
	(*****P13_BottleTransfer********)
	bBottleTransferEnable							:BOOL;(*#p*)         					// Właczenie robota
	nBottleTransferProgram							:UINT;(*#p*)         					// Program robota

 	bBottleTransferDoHoming							:BOOL;									// Rozkaz wykonania pozycjonowania robota
	iBottleTransferPickOffsetX						:INT;
	iBottleTransferPickOffsetY						:INT;  
	iBottleTransferPickOffsetZ						:INT;   
	iBottleTransferPick2OffsetX						:INT;
	iBottleTransferPick2OffsetY						:INT;  
	iBottleTransferPick2OffsetZ						:INT;   

	iBottleTransferPlace1OffsetX					:INT;
	iBottleTransferPlace1OffsetY					:INT;  
	iBottleTransferPlace1OffsetZ					:INT;
	iBottleTransferPlace2OffsetX					:INT;
	iBottleTransferPlace2OffsetY					:INT;
	iBottleTransferPlace2OffsetZ					:INT; 
	iBottleTransferSpeed							:INT := 2;								// predkosc robota pozioma	
	bBottleTransferInkJetEnable						:BOOL;									// Przejazd robota przez InkJet
  	bBottleTransferPickOnlyOne						:BOOL;						// Pobieranie tylko 1 opakowania
	bBottleTransferWeightEnable						:BOOL;
    iBottleTransferWeightInterval					:INT;	
	
	(***P13_BottleTransferAfterDrag***)	
	//Przeciąganie formatek 
	bBottleTransferAfterDragEnable					:BOOL;									// Zezwolenie na pracę przeciągania 
	bBottleTransferAfterDragDoHoming				:BOOL;									// Wykonanie bazowania przeciągania
	bBottleTransferAfterDragHeightSet				:BOOL;									// Wykonanie bazowania przeciągania
		
	(*****P14_BadBottleConyevor********)
	bBadBottleConveyorEnable						:BOOL;									//Zezwolenie na pracę transportera odrzuconych butelek
	nBadBottleConveyorVelocitySV					:UINT;									// Predkosc zadana transportera
	bBadBottleConveyorStart							:BOOL; 									// Zezwolenie na pracę transportera we/wy	

	(*******P14_TurnTable********)
	bExitTurnTableEnable							:BOOL;(**)								//Zezwolenie na pracę etykieciarki
	bExitTurnTableCmdStart 							:BOOL;
	bExitTurnTableGateRun							:BOOL;
	bExitConveyorEnable								:BOOL;(**)								//Zezwolenie na pracę 
	nExitConveyorVelocitySV							:UINT;
	bExitConveyorCmdStart 							:BOOL;
	bExitConveyorGateRun							:BOOL;

	
	(********P15_FormTransporters********)
	bFormTransportersEnable							:BOOL;			
	bFormTransportersDispencerCmdStart				:BOOL; 									// Start transporterów formatek w cyklu
	bFormTransportersBeforeROPPCmdStart				:BOOL;
	bFormTransportersScrewerCmdStart				:BOOL; 									// Start transporterów formatek w cyklu
	bFormTransportersScrewerStop					:BOOL; 									// Start transporterów formatek w cyklu
	bFormTransportersBeforeROPPStop					:BOOL;
	bFormTransportersDispencerSlowSpeedPulse		:BOOL;									// Wolna prędkość transportera
	bFormTransportersDispencerSlowSpeed				:BOOL;									// Wolna prędkość transportera
	bFormTransportersDispencerResetSpeed			:BOOL;									// Reset prędkości transportra
	ulFormTransportersScrewerSlowNumber				:ULINT;									// Nr RFID ostatniej formatki bez korka
	bFormTransportersAfterCapSorterCmdStart			:BOOL;									// Start transportera przez zakręcarka								// Aktywacja
	bFormTransportersBeforeScrewerCmdStart			:BOOL;									// Start transportera przez zakręcarka								// Aktywacja
	bFormTransporterSlowerCmdStart					:BOOL;									// Start transportera spowalniacza fomatek
	bFormTransportersAfterScrewerCmdStart			:BOOL;									// Start transportera przez zakręcarka								// Aktywacja
	ulSingleRealeseIfNoCapFromScrewersNumber		:ULINT;									// Nr RFID ostatniej formatki bez korka
	bSingleRealeseIfNoCapFromScrewersPulse			:BOOL;
	iSingleRealeseIfNoCapFromScrewersPulse			:INT;
				
	//Opcja z falownikiem
	nFormTransportersDispencerVelocitySV			:UDINT;		// Prędkość transportera otwartych butelek
	nFormTransportersScrewerVelocitySV				:UDINT;		// Prędkość transportera zamkniętych butelek
	nFormTransportersAfterCapSorterVelocitySV		:UDINT;		// Prędkość transportera przed zakręcarkami
	nFormTransportersBeforeScrewerVelocitySV		:UDINT;		// Prędkość transportera przed zakręcarkami
	nFormTransportersSlowerVelocitySV				:UDINT;		// Prędkość spowalniacza
	nFormTransportersAfterScrewerVelocitySV			:UDINT;		// Prędkość transportera przed zakręcarkami
	nFormTransportersROPPVelocitySV					:UDINT;		// Prędkość spowalniacza

	(******P16_LabelMachine********)
	bLabelMachineEnable								:BOOL;(**)								//Zezwolenie na pracę etykieciarki
	bLabelMachineCmdStart							:BOOL;		

	(*****P17_CircularInkJet********)
	bCircularInkjetEnable 							:BOOL;									// Zezwolenie na pracę Inkjet'u obwodowego	
	iCircularInkjetSpeed 							:INT;									// Prędkość rolek
	iCircularInkjetDelay							:INT;									// Opóźnienie docisku rolek
	iCircularInkjetHold								:INT;		
	
	bDragingFormsNotDone							:BOOL;				//Zmienna pomocnicza od przeciagania

	(**P20_ExhaustFan**)
	bExhaustFanEnable								:BOOL;
	bExhaustFanCmdStart								:BOOL;
	udiExhaustFanVelocitySV							:UDINT;
	


END_VAR

VAR_GLOBAL PERSISTENT
	(*****Zmienne presistent****)
	
	(***MAIN***)
	eRFID											:ARRAY [1..100] OF S_PackageState;		// STRUKTURA RFID
	AbRFIDFormOrder									:ARRAY [0..100] OF ULINT;				// Globalny rejestr kolejności formatek

	// Auton
	iDispencerRepair1								:INT;
	itonAfterDispencersRepair						:INT;
	itonAfterDispencersRepair1B						:INT;
	itonAfterDispencersRepair2						:INT;	
	itonAfterDispencersRepair3						:INT;	
	itonAfterDispencersRepair4						:INT;	
	itonRobotBottleTransferedToLabelerRepair		:INT;
	itonRobotBottleTransferedToLabeler2Repair		:INT;
	
	(***P00_Counters***)
	nGlobalCounterTemp								:UDINT;									//Tymczasowa zmienna do zapisywania licznika globalnego do pliku raz na jakiś czas
	
	(*Do diagnostyki*)
	iCounterDispencer34DosingAborted				:INT;
	iRepairFormBeforeDispenscerCounter				:INT;
	iRepairFormBeforeDispenscer2PhaseCounter		:INT;
	iRepairAfterDispencerCounter					:INT;
	iRepairBeforeDispencer12Counter					:INT;
	iRepairBeforeDispencer12Counter2				:INT;	
	iWeightRepair1Counter							:INT;
	iWeightRepair2Counter							:INT;
	iRepairFourthFormBeforeDispencerCounter			:INT;
	iRepairBeforeDispencer34Counter					:INT;
	
	iRepairLidFeeder1Counter						:INT;
	iRepairLidFeeder2Counter						:INT;
	iRepairLidFeeder3Counter						:INT;
	iRepairLidFeeder4Counter						:INT;
	
	iUnderScrewerPackageState222nCardNumberChangeCounter		: INT;
	iUnderScrewerPackageState333nCardNumberChangeCounter		: INT;
	iUnderScrewerPackageState111nCardNumberChangeCounter		: INT;
	
	iDispencerPackageState4nCardNumberChangeCounter	:INT;		
	iDispencerPackageState3nCardNumberChangeCounter	:INT;	
	iDispencerPackageState2nCardNumberChangeCounter	:INT;	
	iDispencerPackageState1nCardNumberChangeCounter	:INT;	
	
	iRobotPackageState2nCardNumberChangeCounter		:INT;	
	iRobotPackageState1nCardNumberChangeCounter		:INT;	
	
	iRobotRepairPackageForm1Counter					:INT;
	iRobotRepairPackageForm2Counter					:INT;	
	
	iScrewerFormStuck								:INT;
	iScrewerFormStuck2								:INT;
	iScrewerFormStuck3								:INT;

	(***MAIN***)
	//aSetIDBottle
	nID												:UDINT;									// Identycikacja butelek
		
	(*****P02_Dispencers****)
	bTank1LevelSensorCalibrated						:BOOL;									//Czujnik poziomu nr 1 skalibrowany	
	
	(*****P13_BottleTransfer********)
	nBottleTransferLubricationCounter				:DINT;									//Licznik po którym wyświetla się ostrzeżenie o smarowaniu robota
	
	
END_VAR

(* stored: Version 1.1.0.1, ProductVersion 3.1.4026.13, FileIdentifier 915124c0aa3a7d099c098c68da5dc8adffd3cf0a, FileSignature 2e5229ba9f203ee12088416df98824d7c1d0057249edc83768f87969baed2c69ed3029ca0746e7bfd4beeb3fa4aa8bd0428f18c3a9511c1770b2b46e432803c73bdb8c1e3d73cf75adace2a5c7c1811c7bcce142a4456d5815f6cd2ef5b27e1558c616191c9954f6b86a590d4c45256dea232283c00d16bb937f83ef78d4fb37be567dafd5fb17511a08b04f9c59fdb17056a3918b0f3bfc905bc0c7e1a491c3a4fc408d32179687b55b96b9b2da645b3b837691aca6711b0988fcb1544d8b25463809c9f5721da4ece9298dfd447aa085e8dbb94c5ec692a0a908143da9aac8c1ed607cd6da0202a90d963e93c1b3c7f73e0548fee47b7406d2bf2b220384b7
   GVL GVL: Id {1cf86f2f-5c42-4487-8877-547de30d599a} *)
